{attribute 'linkalways'} 
{attribute 'no_explicit_call' := 'This FB is a CLASS and must be accessed using methods or properties'}
{attribute 'enable_dynamic_creation'}
FUNCTION_BLOCK Node_ContainerType_Vector_UDINT EXTENDS Node
VAR
    out : _GUID;
END_VAR

METHOD PUBLIC  Clone : I_Node
VAR
	pNode : POINTER TO Node_ContainerType_Vector_UDINT;
END_VAR
pNode := __NEW(Node_ContainerType_Vector_UDINT);
Clone := pNode^;
END_METHOD

METHOD FB_init : BOOL
VAR_INPUT
	bInitRetains : BOOL; // if TRUE, the retain variables are initialized (warm start / cold start)
	bInCopyCode : BOOL;  // if TRUE, the instance afterwards gets moved into the copy code (online change)
END_VAR
AddOutput('out', out);
END_METHOD

METHOD PROTECTED OnExecute
out.Value := ContainerType_Vector_UDINT;
END_METHOD

END_FUNCTION_BLOCK

(* stored: Version 1.1.0.1, ProductVersion 3.1.4026.17
   POU Node_ContainerType_Vector_UDINT: Id {7f6a8ef2-1195-019d-05c2-85182e964024}, SpecialFunc None
   Folder Constructor: Id {a144bd0d-936e-0ede-3fc1-7859c860911e}
   Method Clone: Id {352d1274-b815-0ea3-3ffc-d8520d167a8e}
   Method FB_init: Id {256958fd-bbbc-02ae-2942-16d267bdc468}
   Method OnExecute: Id {00949a06-20f8-0e2a-28a5-4c77d3a2c87c} *)
